PROGRAM MAIN
VAR
   i : INT;
END_VAR

i := i + 1;

END_PROGRAM

(* stored: Version 1.1.0.1, ProductVersion 3.1.4024.12
   POU MAIN: Id {7802ecd8-5171-42d6-a8c4-2a1758873295}, SpecialFunc None *)
